// TIA Portal project "MP2019" (V17)

(* hardware
DEVICE "S7-1200 station_1"  S7-1200 Station
   slot 0: "Rack_0"  S7-1200 Rack  Rack  V1.0
   slot 1: "PLC_1"  CPU 1214C DC/DC/DC  6ES7 214-1AG40-0XB0  V4.5
*)

// ===== PLC "PLC_1"  CPU 1214C DC/DC/DC =====

VAR_GLOBAL   // PLC tag table "Default tag table"
   "wysoki_poziom" AT %I0.1 : Bool;
   "Tag_2" AT %I0.2 : Bool;
   "pompa_1" AT %Q0.0 : Bool;
   "pompa_2" AT %Q0.1 : Bool;
   "Tag_5" AT %M50.0 : Bool;
   "Tag_6" AT %M50.1 : Bool;
   "Tag_7" AT %M50.2 : Bool;
   "Tag_8" AT %M50.3 : Bool;
   "niski_poziom" AT %I0.0 : Bool;
   "Tag_10" AT %Q0.3 : Bool;
   "Tag_11" AT %I0.3 : Bool;
   "Tag_12" AT %Q0.4 : Bool;
   "Tag_13" AT %Q0.5 : Bool;
   "Tag_14" AT %Q0.6 : Bool;
   "Tag_15" AT %IW64 : Int;
   "Clock_Byte" AT %MB0 : Byte;
   "Clock_10Hz" AT %M0.0 : Bool;
   "Clock_5Hz" AT %M0.1 : Bool;
   "Clock_2.5Hz" AT %M0.2 : Bool;
   "Clock_2Hz" AT %M0.3 : Bool;
   "Clock_1.25Hz" AT %M0.4 : Bool;
   "Clock_1Hz" AT %M0.5 : Bool;
   "Clock_0.625Hz" AT %M0.6 : Bool;
   "Clock_0.5Hz" AT %M0.7 : Bool;
   "alarm" AT %Q0.7 : Bool;
   "Tag_1" AT %I0.7 : Bool;
END_VAR

DATA_BLOCK "grupowe1_DB"   // DB1
{ S7_Optimized_Access := 'TRUE' }
VERSION : 0.1
// stored: InstanceOfName grupowe1
"grupowe1"
BEGIN
END_DATA_BLOCK

DATA_BLOCK "grupowe2_DB"   // DB2
{ S7_Optimized_Access := 'TRUE' }
VERSION : 0.1
// stored: InstanceOfName grupowe2
"grupowe2"
BEGIN
END_DATA_BLOCK

DATA_BLOCK "grupowe4_DB"   // DB8
{ S7_Optimized_Access := 'TRUE' }
VERSION : 0.1
// stored: InstanceOfName grupowe4
"grupowe4"
BEGIN
END_DATA_BLOCK

DATA_BLOCK "grupowe6_DB"   // DB9
{ S7_Optimized_Access := 'TRUE' }
VERSION : 0.1
// stored: InstanceOfName grupowe6
"grupowe6"
BEGIN
END_DATA_BLOCK

DATA_BLOCK "grupowe7_DB"   // DB13
{ S7_Optimized_Access := 'TRUE' }
VERSION : 0.1
// stored: InstanceOfName grupowe7
"grupowe7"
BEGIN
END_DATA_BLOCK

DATA_BLOCK "final_Master_DB"   // DB14
{ S7_Optimized_Access := 'TRUE' }
VERSION : 0.1
// stored: InstanceOfName final_Master
"final_Master"
BEGIN
END_DATA_BLOCK

DATA_BLOCK "final_Ekspert_DB"   // DB15
{ S7_Optimized_Access := 'TRUE' }
VERSION : 0.1
// stored: InstanceOfName final_Ekspert
"final_Ekspert"
BEGIN
END_DATA_BLOCK

// folder: System blocks/Program resources

DATA_BLOCK "IEC_Timer_0_DB"   // DB3
{ S7_Optimized_Access := 'TRUE' }
AUTHOR : Simatic
FAMILY : IEC
NAME : IEC_TMR
VERSION : 1.0
// stored: InstanceOfName IEC_TIMER
"IEC_TIMER"
BEGIN
END_DATA_BLOCK

DATA_BLOCK "IEC_Timer_0_DB_1"   // DB4
{ S7_Optimized_Access := 'TRUE' }
AUTHOR : Simatic
FAMILY : IEC
NAME : IEC_TMR
VERSION : 1.0
// stored: InstanceOfName IEC_TIMER
"IEC_TIMER"
BEGIN
END_DATA_BLOCK

DATA_BLOCK "Counter0"   // DB5
{ S7_Optimized_Access := 'TRUE' }
AUTHOR : Simatic
FAMILY : IEC
NAME : CNTR
VERSION : 1.0
// stored: InstanceOfName IEC_COUNTER
"IEC_COUNTER"
BEGIN
END_DATA_BLOCK

DATA_BLOCK "IEC_Timer_0_DB_3"   // DB6
{ S7_Optimized_Access := 'TRUE' }
AUTHOR : Simatic
FAMILY : IEC
NAME : IEC_TMR
VERSION : 1.0
// stored: InstanceOfName IEC_TIMER
"IEC_TIMER"
BEGIN
END_DATA_BLOCK

DATA_BLOCK "IEC_Timer_0_DB_4"   // DB7
{ S7_Optimized_Access := 'TRUE' }
AUTHOR : Simatic
FAMILY : IEC
NAME : IEC_TMR
VERSION : 1.0
// stored: InstanceOfName IEC_TIMER
"IEC_TIMER"
BEGIN
END_DATA_BLOCK

DATA_BLOCK "TON0"   // DB10
{ S7_Optimized_Access := 'TRUE' }
AUTHOR : Simatic
FAMILY : IEC
NAME : IEC_TMR
VERSION : 1.0
// stored: InstanceOfName IEC_TIMER
"IEC_TIMER"
BEGIN
END_DATA_BLOCK

DATA_BLOCK "TON1"   // DB11
{ S7_Optimized_Access := 'TRUE' }
AUTHOR : Simatic
FAMILY : IEC
NAME : IEC_TMR
VERSION : 1.0
// stored: InstanceOfName IEC_TIMER
"IEC_TIMER"
BEGIN
END_DATA_BLOCK

DATA_BLOCK "TON2"   // DB12
{ S7_Optimized_Access := 'TRUE' }
AUTHOR : Simatic
FAMILY : IEC
NAME : IEC_TMR
VERSION : 1.0
// stored: InstanceOfName IEC_TIMER
"IEC_TIMER"
BEGIN
END_DATA_BLOCK

// folder: (top level)

FUNCTION_BLOCK "grupowe1"   // FB1, LAD
{ S7_Optimized_Access := 'TRUE' }
VERSION : 0.1
   VAR_INPUT
      IN1 : Bool;
      IN2 : Bool;
   END_VAR
   VAR_IN_OUT
      OUT0 : Bool;
      OUT1 : Bool;
   END_VAR
   VAR
      IN1_edge : Bool;
      IN2_edge : Bool;
   END_VAR
   VAR_TEMP
      prev_OUT0 : Bool;
      prev_OUT1 : Bool;
   END_VAR
   VAR_TEMP   // added for the SCL form of the ladder/FBD networks
      _w1 : Bool;
   END_VAR
BEGIN

REGION Network 1
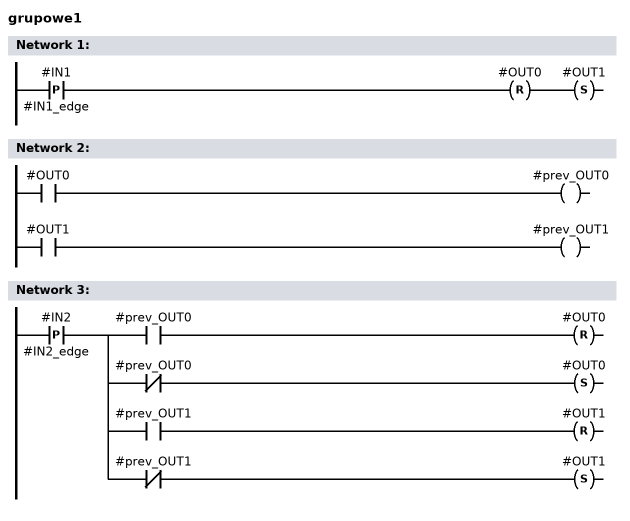
   RUNG wire#powerrail
      P_Contact(operand := #IN1, bit := #IN1_edge)
      R_Coil( #OUT0 )
      S_Coil( #OUT1 )
   END_RUNG
   // the same network as SCL:
   #_w1 := #IN1 AND NOT #IN1_edge;   // rising edge of #IN1
   #IN1_edge := #IN1;
   IF #_w1 THEN
       #OUT0 := FALSE;
       #OUT1 := TRUE;
   END_IF;
END_REGION

REGION Network 2
   RUNG wire#powerrail
      Contact( #OUT0 )
      Coil( #prev_OUT0 )
   END_RUNG
   RUNG wire#powerrail
      Contact( #OUT1 )
      Coil( #prev_OUT1 )
   END_RUNG
   // the same network as SCL:
   #prev_OUT0 := #OUT0;
   #prev_OUT1 := #OUT1;
END_REGION

REGION Network 3
   RUNG wire#powerrail
      P_Contact(operand := #IN2, bit := #IN2_edge)
      wire#w1
      Contact( #prev_OUT0 )
      R_Coil( #OUT0 )
   END_RUNG
   RUNG wire#w1
      I_Contact( #prev_OUT0 )
      S_Coil( #OUT0 )
   END_RUNG
   RUNG wire#w1
      Contact( #prev_OUT1 )
      R_Coil( #OUT1 )
   END_RUNG
   RUNG wire#w1
      I_Contact( #prev_OUT1 )
      S_Coil( #OUT1 )
   END_RUNG
   // the same network as SCL:
   #_w1 := #IN2 AND NOT #IN2_edge;   // rising edge of #IN2
   #IN2_edge := #IN2;
   IF #_w1 AND #prev_OUT0 THEN #OUT0 := FALSE; END_IF;
   IF #_w1 AND NOT #prev_OUT0 THEN #OUT0 := TRUE; END_IF;
   IF #_w1 AND #prev_OUT1 THEN #OUT1 := FALSE; END_IF;
   IF #_w1 AND NOT #prev_OUT1 THEN #OUT1 := TRUE; END_IF;
END_REGION
END_FUNCTION_BLOCK

FUNCTION_BLOCK "grupowe2"   // FB2, LAD
{ S7_Optimized_Access := 'TRUE' }
VERSION : 0.1
   VAR_INPUT
      IN2 : Bool;
      IN3 : Bool;
   END_VAR
   VAR_IN_OUT
      OUT3 : Bool;
   END_VAR
   VAR
      IN2_edge : Bool;
      IN3_edge : Bool;
      step1 : Bool;
   END_VAR
   VAR_TEMP
      prev_OUT3 : Bool;
   END_VAR
   VAR_TEMP   // added for the SCL form of the ladder/FBD networks
      _w1 : Bool;
      _w2 : Bool;
   END_VAR
BEGIN

REGION Network 1
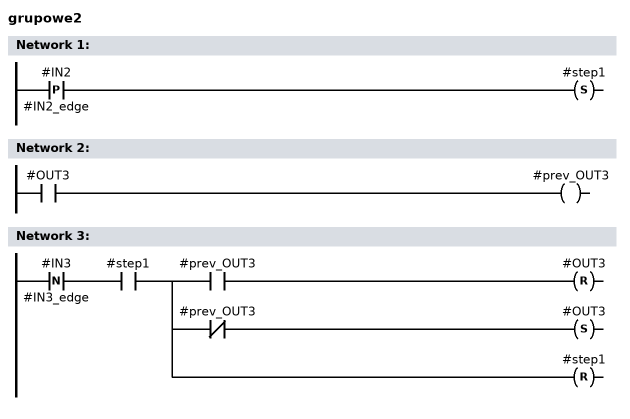
   RUNG wire#powerrail
      P_Contact(operand := #IN2, bit := #IN2_edge)
      S_Coil( #step1 )
   END_RUNG
   // the same network as SCL:
   #_w1 := #IN2 AND NOT #IN2_edge;   // rising edge of #IN2
   #IN2_edge := #IN2;
   IF #_w1 THEN #step1 := TRUE; END_IF;
END_REGION

REGION Network 2
   RUNG wire#powerrail
      Contact( #OUT3 )
      Coil( #prev_OUT3 )
   END_RUNG
   // the same network as SCL:
   #prev_OUT3 := #OUT3;
END_REGION

REGION Network 3
   RUNG wire#powerrail
      N_Contact(operand := #IN3, bit := #IN3_edge)
      Contact( #step1 )
      wire#w1
      Contact( #prev_OUT3 )
      R_Coil( #OUT3 )
   END_RUNG
   RUNG wire#w1
      I_Contact( #prev_OUT3 )
      S_Coil( #OUT3 )
   END_RUNG
   RUNG wire#w1
      R_Coil( #step1 )
   END_RUNG
   // the same network as SCL:
   #_w1 := NOT #IN3 AND #IN3_edge;   // falling edge of #IN3
   #IN3_edge := #IN3;
   #_w2 := #_w1 AND #step1;
   IF #_w2 AND #prev_OUT3 THEN #OUT3 := FALSE; END_IF;
   IF #_w2 AND NOT #prev_OUT3 THEN #OUT3 := TRUE; END_IF;
   IF #_w2 THEN #step1 := FALSE; END_IF;
END_REGION
END_FUNCTION_BLOCK

FUNCTION_BLOCK "grupowe4"   // FB3, LAD
{ S7_Optimized_Access := 'TRUE' }
VERSION : 0.1
   VAR_INPUT
      IN2 : Bool;
   END_VAR
   VAR_OUTPUT
      OUT : Bool;
   END_VAR
BEGIN

REGION Network 1
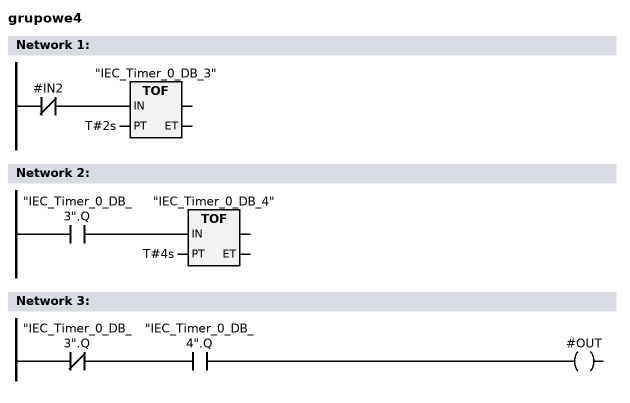
   "IEC_Timer_0_DB_3".TOF(IN := NOT #IN2, PT := T#2s);
END_REGION

REGION Network 2
   "IEC_Timer_0_DB_4".TOF(IN := "IEC_Timer_0_DB_3".Q, PT := T#4s);
END_REGION

REGION Network 3
   RUNG wire#powerrail
      I_Contact( "IEC_Timer_0_DB_3".Q )
      Contact( "IEC_Timer_0_DB_4".Q )
      Coil( #OUT )
   END_RUNG
   // the same network as SCL:
   #OUT := NOT "IEC_Timer_0_DB_3".Q AND "IEC_Timer_0_DB_4".Q;
END_REGION
END_FUNCTION_BLOCK

FUNCTION_BLOCK "grupowe6"   // FB4, LAD
{ S7_Optimized_Access := 'TRUE' }
VERSION : 0.1
   VAR_INPUT
      IN2 : Bool;
      IN3 : Bool;
   END_VAR
   VAR_OUTPUT
      OUT0 : Bool;
   END_VAR
   VAR_IN_OUT
      Value : Int;
   END_VAR
   VAR
      IN2_edge : Bool;
      IN3_edge : Bool;
   END_VAR
   VAR_TEMP
      Modulo : USInt;
   END_VAR
   VAR_TEMP   // added for the SCL form of the ladder/FBD networks
      _w1 : Bool;
      _w2 : Bool;
   END_VAR
BEGIN

REGION Network 1
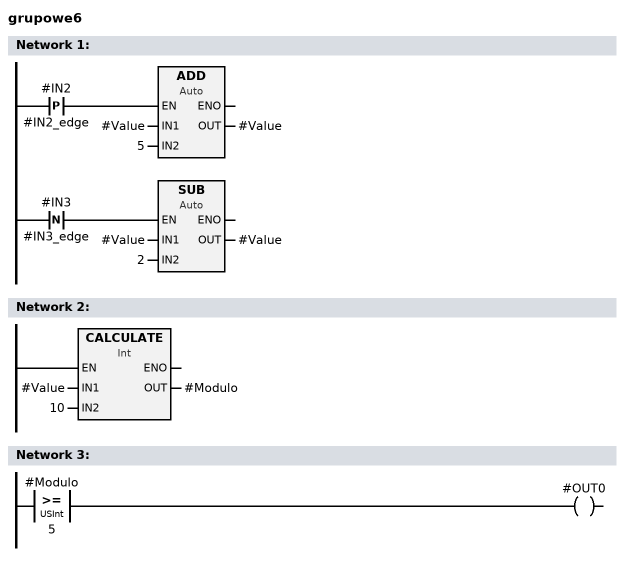
   RUNG wire#powerrail
      P_Contact(operand := #IN2, bit := #IN2_edge)
      Add(in1 := #Value, in2 := 5, out => #Value)
   END_RUNG
   RUNG wire#powerrail
      N_Contact(operand := #IN3, bit := #IN3_edge)
      Sub(in1 := #Value, in2 := 2, out => #Value)
   END_RUNG
   // the same network as SCL:
   #_w1 := #IN2 AND NOT #IN2_edge;   // rising edge of #IN2
   #IN2_edge := #IN2;
   IF #_w1 THEN #Value := #Value + 5; END_IF;
   #_w2 := NOT #IN3 AND #IN3_edge;   // falling edge of #IN3
   #IN3_edge := #IN3;
   IF #_w2 THEN #Value := #Value - 2; END_IF;
END_REGION

REGION Network 2
   RUNG wire#powerrail
      { S7_Templates := "SrcType := Int"; S7_Expression := "IN1 MOD IN2" } Calculate(in1 := #Value, in2 := 10, out => #Modulo)
   END_RUNG
   // the same network as SCL:
   #Modulo := #Value MOD 10;
END_REGION

REGION Network 3
   RUNG wire#powerrail
      { S7_Templates := "SrcType := USInt" } GE_Contact(in1 := #Modulo, in2 := 5)
      Coil( #OUT0 )
   END_RUNG
   // the same network as SCL:
   #OUT0 := #Modulo >= 5;
END_REGION
END_FUNCTION_BLOCK

FUNCTION_BLOCK "grupowe7"   // FB5, LAD
{ S7_Optimized_Access := 'TRUE' }
VERSION : 0.1
   VAR_INPUT
      Analog_signal : Int;
   END_VAR
   VAR_OUTPUT
      OUT0 : Bool;
      OUT4 : Bool;
      OUT5 : Bool;
      OUT6 : Bool;
   END_VAR
   VAR
      TON0_Q : Bool;
   END_VAR
   VAR_TEMP
      duty : Int;
      Analog_norm : Real;
      T_high : DInt;
      Hz : Bool;
   END_VAR
BEGIN

REGION Network 1
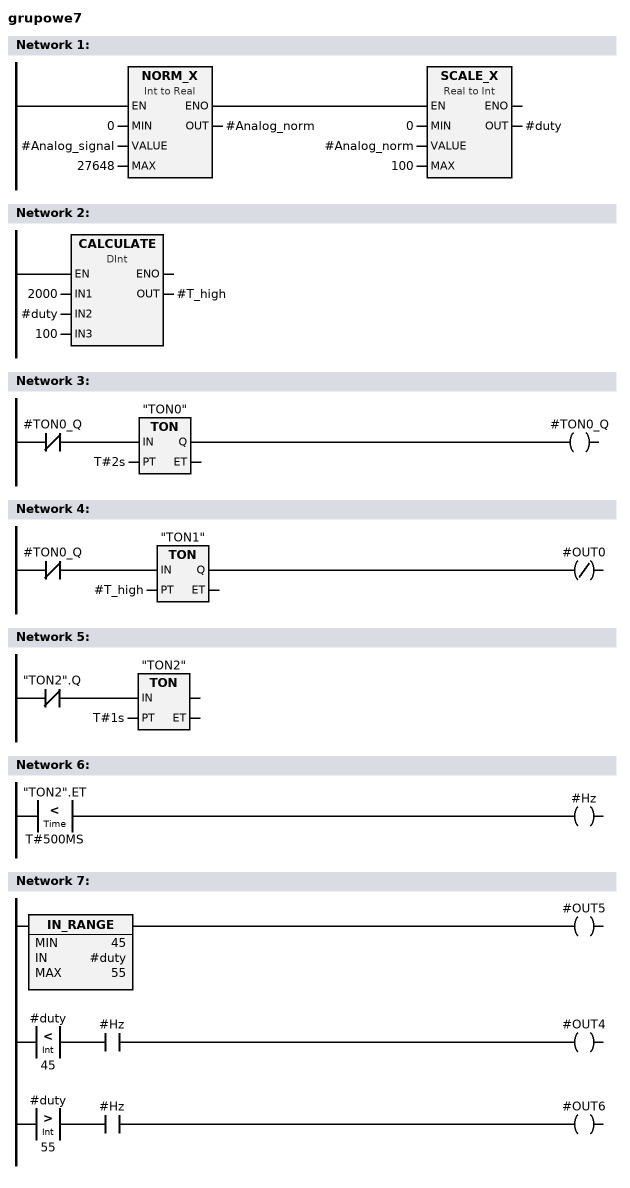
   RUNG wire#powerrail
      { S7_Templates := "[SrcType := Int, DestType := Real]" } Normalize(min := 0, value := #Analog_signal, max := 27648, out => #Analog_norm)
      { S7_Templates := "[SrcType := Real, DestType := Int]" } Scale(min := 0, value := #Analog_norm, max := 100, out => #duty)
   END_RUNG
   // the same network as SCL:
   #Analog_norm := NORM_X(MIN := 0, VALUE := #Analog_signal, MAX := 27648);
   #duty := SCALE_X(MIN := 0, VALUE := #Analog_norm, MAX := 100);
END_REGION

REGION Network 2
   RUNG wire#powerrail
      { S7_Templates := "SrcType := DInt"; S7_Expression := "IN1 * IN2 / IN3" } Calculate(in1 := 2000, in2 := #duty, in3 := 100, out => #T_high)
   END_RUNG
   // the same network as SCL:
   #T_high := 2000 * #duty / 100;
END_REGION

REGION Network 3
   "TON0".TON(IN := NOT #TON0_Q, PT := T#2s);
   #TON0_Q := "TON0".Q;
END_REGION

REGION Network 4
   "TON1".TON(IN := NOT #TON0_Q, PT := #T_high);
   #OUT0 := NOT "TON1".Q;
END_REGION

REGION Network 5
   "TON2".TON(IN := NOT "TON2".Q, PT := T#1s);
END_REGION

REGION Network 6
   RUNG wire#powerrail
      { S7_Templates := "SrcType := Time" } LT_Contact(in1 := "TON2".ET, in2 := T#500MS)
      Coil( #Hz )
   END_RUNG
   // the same network as SCL:
   #Hz := "TON2".ET < T#500MS;
END_REGION

REGION Network 7
   RUNG wire#powerrail
      { S7_Templates := "SrcType := Int" } InRange(min := 45, in := #duty, max := 55)
      Coil( #OUT5 )
   END_RUNG
   RUNG wire#powerrail
      { S7_Templates := "SrcType := Int" } LT_Contact(in1 := #duty, in2 := 45)
      Contact( #Hz )
      Coil( #OUT4 )
   END_RUNG
   RUNG wire#powerrail
      { S7_Templates := "SrcType := Int" } GT_Contact(in1 := #duty, in2 := 55)
      Contact( #Hz )
      Coil( #OUT6 )
   END_RUNG
   // the same network as SCL:
   #OUT5 := (45 <= #duty) AND (#duty <= 55);
   #OUT4 := (#duty < 45) AND #Hz;
   #OUT6 := (#duty > 55) AND #Hz;
END_REGION
END_FUNCTION_BLOCK

FUNCTION_BLOCK "final_Master"   // FB6, LAD
{ S7_Optimized_Access := 'TRUE' }
VERSION : 0.1
   VAR_INPUT
      niski_poziom : Bool;
      wysoki_poziom : Bool;
   END_VAR
   VAR_OUTPUT
      alarm : Bool;
      segment1 : Bool;
      segment2 : Bool;
      segment4 : Bool;
   END_VAR
   VAR_IN_OUT
      pompa_1 : Bool;
      pompa_2 : Bool;
   END_VAR
   VAR
      niski_zbocze : Bool;
      wysoki_zbocze : Bool;
      pompa_ostatnio : Bool;
      niski_zbocze2 : Bool;
      wysoki_zbocze2 : Bool;
      prev_pompa : Bool;
   END_VAR
   VAR_TEMP   // added for the SCL form of the ladder/FBD networks
      _w1 : Bool;
      _w2 : Bool;
      _w3 : Bool;
   END_VAR
BEGIN

REGION Network 1
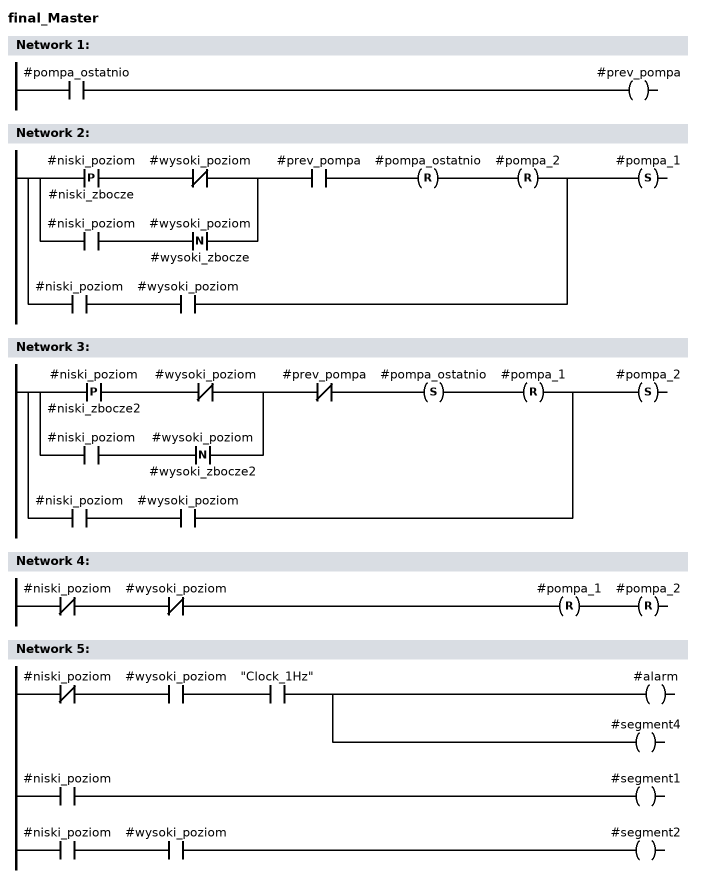
   RUNG wire#powerrail
      Contact( #pompa_ostatnio )
      Coil( #prev_pompa )
   END_RUNG
   // the same network as SCL:
   #prev_pompa := #pompa_ostatnio;
END_REGION

REGION Network 2
   RUNG wire#powerrail
      P_Contact(operand := #niski_poziom, bit := #niski_zbocze)
      I_Contact( #wysoki_poziom )
      wire#w1
      Contact( #prev_pompa )
      R_Coil( #pompa_ostatnio )
      R_Coil( #pompa_2 )
      wire#w2
      S_Coil( #pompa_1 )
   END_RUNG
   RUNG wire#powerrail
      Contact( #niski_poziom )
      N_Contact(operand := #wysoki_poziom, bit := #wysoki_zbocze)
   END_RUNG wire#w1
   RUNG wire#powerrail
      Contact( #niski_poziom )
      Contact( #wysoki_poziom )
   END_RUNG wire#w2
   // the same network as SCL:
   #_w1 := #niski_poziom AND NOT #niski_zbocze;   // rising edge of #niski_poziom
   #niski_zbocze := #niski_poziom;
   #_w2 := #niski_poziom AND NOT #wysoki_poziom AND #wysoki_zbocze;   // falling edge of #wysoki_poziom
   #wysoki_zbocze := #wysoki_poziom;
   #_w3 := ((#_w1 AND NOT #wysoki_poziom) OR #_w2) AND #prev_pompa;
   IF #_w3 THEN
       #pompa_ostatnio := FALSE;
       #pompa_2 := FALSE;
   END_IF;
   IF #_w3 OR (#niski_poziom AND #wysoki_poziom) THEN #pompa_1 := TRUE; END_IF;
END_REGION

REGION Network 3
   RUNG wire#powerrail
      P_Contact(operand := #niski_poziom, bit := #niski_zbocze2)
      I_Contact( #wysoki_poziom )
      wire#w1
      I_Contact( #prev_pompa )
      S_Coil( #pompa_ostatnio )
      R_Coil( #pompa_1 )
      wire#w2
      S_Coil( #pompa_2 )
   END_RUNG
   RUNG wire#powerrail
      Contact( #niski_poziom )
      N_Contact(operand := #wysoki_poziom, bit := #wysoki_zbocze2)
   END_RUNG wire#w1
   RUNG wire#powerrail
      Contact( #niski_poziom )
      Contact( #wysoki_poziom )
   END_RUNG wire#w2
   // the same network as SCL:
   #_w1 := #niski_poziom AND NOT #niski_zbocze2;   // rising edge of #niski_poziom
   #niski_zbocze2 := #niski_poziom;
   #_w2 := #niski_poziom AND NOT #wysoki_poziom AND #wysoki_zbocze2;   // falling edge of #wysoki_poziom
   #wysoki_zbocze2 := #wysoki_poziom;
   #_w3 := ((#_w1 AND NOT #wysoki_poziom) OR #_w2) AND NOT #prev_pompa;
   IF #_w3 THEN
       #pompa_ostatnio := TRUE;
       #pompa_1 := FALSE;
   END_IF;
   IF #_w3 OR (#niski_poziom AND #wysoki_poziom) THEN #pompa_2 := TRUE; END_IF;
END_REGION

REGION Network 4
   RUNG wire#powerrail
      I_Contact( #niski_poziom )
      I_Contact( #wysoki_poziom )
      R_Coil( #pompa_1 )
      R_Coil( #pompa_2 )
   END_RUNG
   // the same network as SCL:
   IF NOT #niski_poziom AND NOT #wysoki_poziom THEN
       #pompa_1 := FALSE;
       #pompa_2 := FALSE;
   END_IF;
END_REGION

REGION Network 5
   RUNG wire#powerrail
      I_Contact( #niski_poziom )
      Contact( #wysoki_poziom )
      Contact( "Clock_1Hz" )
      wire#w1
      Coil( #alarm )
   END_RUNG
   RUNG wire#w1
      Coil( #segment4 )
   END_RUNG
   RUNG wire#powerrail
      Contact( #niski_poziom )
      Coil( #segment1 )
   END_RUNG
   RUNG wire#powerrail
      Contact( #niski_poziom )
      Contact( #wysoki_poziom )
      Coil( #segment2 )
   END_RUNG
   // the same network as SCL:
   #alarm := NOT #niski_poziom AND #wysoki_poziom AND "Clock_1Hz";
   #segment4 := #alarm;
   #segment1 := #niski_poziom;
   #segment2 := #niski_poziom AND #wysoki_poziom;
END_REGION
END_FUNCTION_BLOCK

FUNCTION_BLOCK "final_Ekspert"   // FB7, LAD
{ S7_Optimized_Access := 'TRUE' }
VERSION : 0.1
   VAR_INPUT
      niski_poziom : Bool;
      wysoki_poziom : Bool;
      tryb_pracy_zmiana : Bool;
   END_VAR
   VAR_OUTPUT
      alarm : Bool;
      segment1 : Bool;
      segment2 : Bool;
      segment4 : Bool;
   END_VAR
   VAR_IN_OUT
      pompa_1 : Bool;
      tryb_pracy : Int;
      pompa_2 : Bool;
   END_VAR
   VAR
      niski_zbocze : Bool;
      wysoki_zbocze : Bool;
      pompa_ostatnio : Bool;
      niski_zbocze2 : Bool;
      wysoki_zbocze2 : Bool;
      prev_pompa : Bool;
      tryb_pracy_zboczeP : Bool;
      tryb_pracy_zboczeN : Bool;
   END_VAR
   VAR_TEMP   // added for the SCL form of the ladder/FBD networks
      _w1 : Bool;
      _w2 : Bool;
      _w3 : Bool;
      _w4 : Bool;
   END_VAR
BEGIN

REGION Network 1
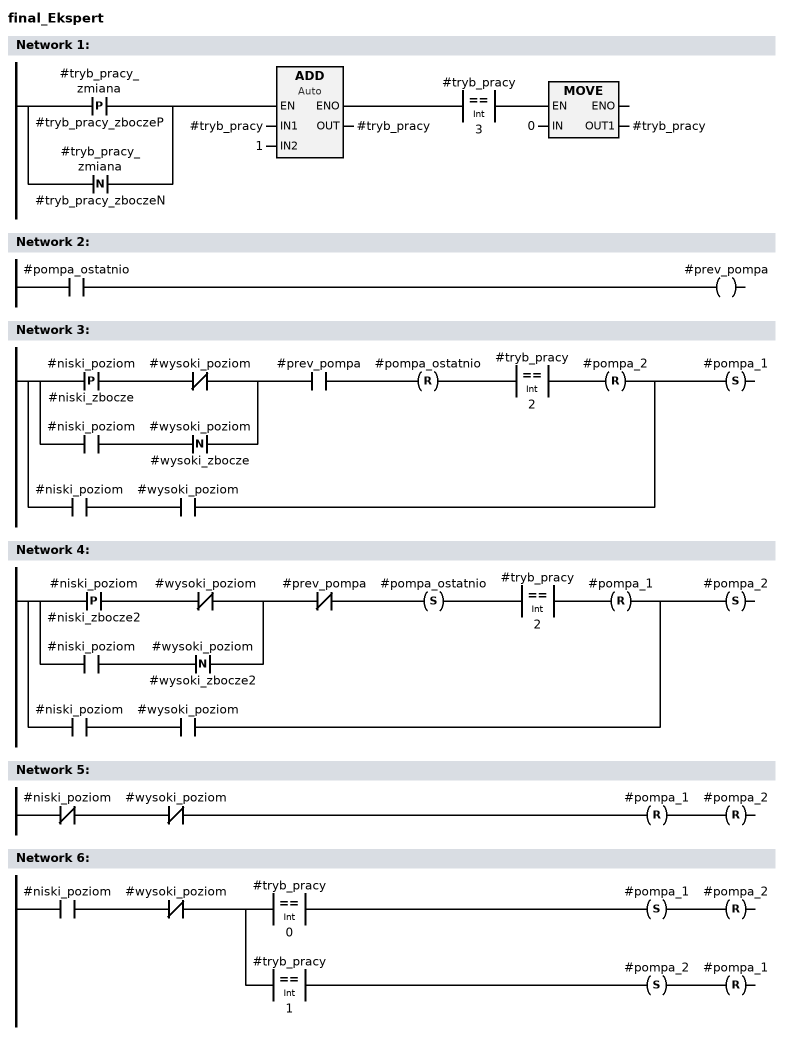
   RUNG wire#powerrail
      P_Contact(operand := #tryb_pracy_zmiana, bit := #tryb_pracy_zboczeP)
      wire#w1
      Add(in1 := #tryb_pracy, in2 := 1, out => #tryb_pracy)
      { S7_Templates := "SrcType := Int" } EQ_Contact(in1 := #tryb_pracy, in2 := 3)
      Move(in := 0, out1 => #tryb_pracy)
   END_RUNG
   RUNG wire#powerrail
      N_Contact(operand := #tryb_pracy_zmiana, bit := #tryb_pracy_zboczeN)
   END_RUNG wire#w1
   // the same network as SCL:
   #_w1 := #tryb_pracy_zmiana AND NOT #tryb_pracy_zboczeP;   // rising edge of #tryb_pracy_zmiana
   #tryb_pracy_zboczeP := #tryb_pracy_zmiana;
   #_w2 := NOT #tryb_pracy_zmiana AND #tryb_pracy_zboczeN;   // falling edge of #tryb_pracy_zmiana
   #tryb_pracy_zboczeN := #tryb_pracy_zmiana;
   #_w3 := #_w1 OR #_w2;
   IF #_w3 THEN #tryb_pracy := #tryb_pracy + 1; END_IF;
   IF #_w3 AND (#tryb_pracy = 3) THEN #tryb_pracy := 0; END_IF;
END_REGION

REGION Network 2
   RUNG wire#powerrail
      Contact( #pompa_ostatnio )
      Coil( #prev_pompa )
   END_RUNG
   // the same network as SCL:
   #prev_pompa := #pompa_ostatnio;
END_REGION

REGION Network 3
   RUNG wire#powerrail
      P_Contact(operand := #niski_poziom, bit := #niski_zbocze)
      I_Contact( #wysoki_poziom )
      wire#w1
      Contact( #prev_pompa )
      R_Coil( #pompa_ostatnio )
      { S7_Templates := "SrcType := Int" } EQ_Contact(in1 := #tryb_pracy, in2 := 2)
      R_Coil( #pompa_2 )
      wire#w2
      S_Coil( #pompa_1 )
   END_RUNG
   RUNG wire#powerrail
      Contact( #niski_poziom )
      N_Contact(operand := #wysoki_poziom, bit := #wysoki_zbocze)
   END_RUNG wire#w1
   RUNG wire#powerrail
      Contact( #niski_poziom )
      Contact( #wysoki_poziom )
   END_RUNG wire#w2
   // the same network as SCL:
   #_w1 := #niski_poziom AND NOT #niski_zbocze;   // rising edge of #niski_poziom
   #niski_zbocze := #niski_poziom;
   #_w2 := #niski_poziom AND NOT #wysoki_poziom AND #wysoki_zbocze;   // falling edge of #wysoki_poziom
   #wysoki_zbocze := #wysoki_poziom;
   #_w3 := ((#_w1 AND NOT #wysoki_poziom) OR #_w2) AND #prev_pompa;
   IF #_w3 THEN #pompa_ostatnio := FALSE; END_IF;
   #_w4 := #_w3 AND (#tryb_pracy = 2);
   IF #_w4 THEN #pompa_2 := FALSE; END_IF;
   IF #_w4 OR (#niski_poziom AND #wysoki_poziom) THEN #pompa_1 := TRUE; END_IF;
END_REGION

REGION Network 4
   RUNG wire#powerrail
      P_Contact(operand := #niski_poziom, bit := #niski_zbocze2)
      I_Contact( #wysoki_poziom )
      wire#w1
      I_Contact( #prev_pompa )
      S_Coil( #pompa_ostatnio )
      { S7_Templates := "SrcType := Int" } EQ_Contact(in1 := #tryb_pracy, in2 := 2)
      R_Coil( #pompa_1 )
      wire#w2
      S_Coil( #pompa_2 )
   END_RUNG
   RUNG wire#powerrail
      Contact( #niski_poziom )
      N_Contact(operand := #wysoki_poziom, bit := #wysoki_zbocze2)
   END_RUNG wire#w1
   RUNG wire#powerrail
      Contact( #niski_poziom )
      Contact( #wysoki_poziom )
   END_RUNG wire#w2
   // the same network as SCL:
   #_w1 := #niski_poziom AND NOT #niski_zbocze2;   // rising edge of #niski_poziom
   #niski_zbocze2 := #niski_poziom;
   #_w2 := #niski_poziom AND NOT #wysoki_poziom AND #wysoki_zbocze2;   // falling edge of #wysoki_poziom
   #wysoki_zbocze2 := #wysoki_poziom;
   #_w3 := ((#_w1 AND NOT #wysoki_poziom) OR #_w2) AND NOT #prev_pompa;
   IF #_w3 THEN #pompa_ostatnio := TRUE; END_IF;
   #_w4 := #_w3 AND (#tryb_pracy = 2);
   IF #_w4 THEN #pompa_1 := FALSE; END_IF;
   IF #_w4 OR (#niski_poziom AND #wysoki_poziom) THEN #pompa_2 := TRUE; END_IF;
END_REGION

REGION Network 5
   RUNG wire#powerrail
      I_Contact( #niski_poziom )
      I_Contact( #wysoki_poziom )
      R_Coil( #pompa_1 )
      R_Coil( #pompa_2 )
   END_RUNG
   // the same network as SCL:
   IF NOT #niski_poziom AND NOT #wysoki_poziom THEN
       #pompa_1 := FALSE;
       #pompa_2 := FALSE;
   END_IF;
END_REGION

REGION Network 6
   RUNG wire#powerrail
      Contact( #niski_poziom )
      I_Contact( #wysoki_poziom )
      wire#w1
      { S7_Templates := "SrcType := Int" } EQ_Contact(in1 := #tryb_pracy, in2 := 0)
      S_Coil( #pompa_1 )
      R_Coil( #pompa_2 )
   END_RUNG
   RUNG wire#w1
      { S7_Templates := "SrcType := Int" } EQ_Contact(in1 := #tryb_pracy, in2 := 1)
      S_Coil( #pompa_2 )
      R_Coil( #pompa_1 )
   END_RUNG
   // the same network as SCL:
   #_w1 := #niski_poziom AND NOT #wysoki_poziom;
   IF #_w1 AND (#tryb_pracy = 0) THEN
       #pompa_1 := TRUE;
       #pompa_2 := FALSE;
   END_IF;
   IF #_w1 AND (#tryb_pracy = 1) THEN
       #pompa_2 := TRUE;
       #pompa_1 := FALSE;
   END_IF;
END_REGION
END_FUNCTION_BLOCK

FUNCTION "grupowe3" : Void   // FC1, LAD
{ S7_Optimized_Access := 'TRUE' }
VERSION : 0.1
   VAR_INPUT
      f : Real;
      duty : Int;
   END_VAR
   VAR_OUTPUT
      OUT : Bool;
   END_VAR
   VAR_TEMP
      T : DInt;
      T_Real : Real;
      T_high : DInt;
   END_VAR
BEGIN

REGION Network 1
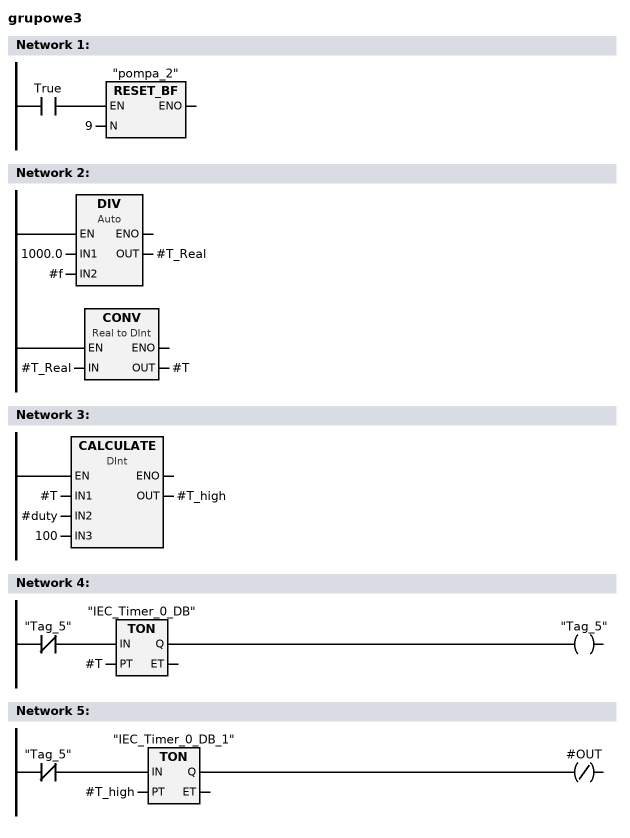
   // no SCL statement known for RBitfield: written as a call
   IF True THEN RESET_BF(operand := "pompa_2", n := 9); END_IF;
END_REGION

REGION Network 2
   RUNG wire#powerrail
      Div(in1 := 1000.0, in2 := #f, out => #T_Real)
   END_RUNG
   RUNG wire#powerrail
      { S7_Templates := "[SrcType := Real, DestType := DInt]" } Convert(in := #T_Real, out => #T)
   END_RUNG
   // the same network as SCL:
   #T_Real := 1000.0 / #f;
   #T := REAL_TO_DINT(#T_Real);
END_REGION

REGION Network 3
   RUNG wire#powerrail
      { S7_Templates := "SrcType := DInt"; S7_Expression := "IN1*IN2/IN3" } Calculate(in1 := #T, in2 := #duty, in3 := 100, out => #T_high)
   END_RUNG
   // the same network as SCL:
   #T_high := #T*#duty/100;
END_REGION

REGION Network 4
   "IEC_Timer_0_DB".TON(IN := NOT "Tag_5", PT := #T);
   "Tag_5" := "IEC_Timer_0_DB".Q;
END_REGION

REGION Network 5
   "IEC_Timer_0_DB_1".TON(IN := NOT "Tag_5", PT := #T_high);
   #OUT := NOT "IEC_Timer_0_DB_1".Q;
END_REGION
END_FUNCTION

FUNCTION "grupowe5" : Void   // FC2, LAD
{ S7_Optimized_Access := 'TRUE' }
VERSION : 0.1
   VAR_INPUT
      IN : Bool;
   END_VAR
   VAR_OUTPUT
      OUT : Bool;
   END_VAR
   VAR_TEMP
      Mod_result : Int;
   END_VAR
BEGIN

REGION Network 1
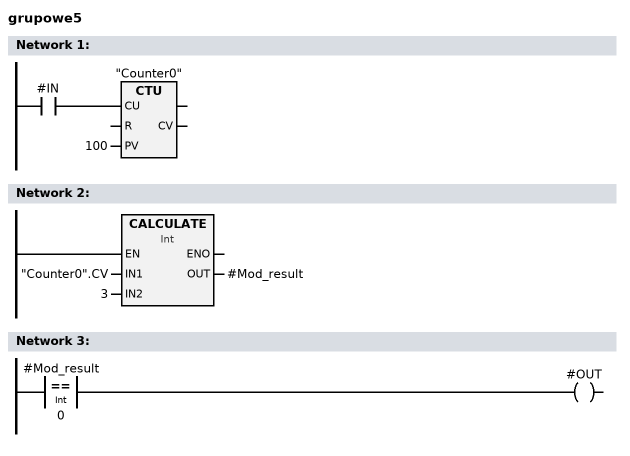
   "Counter0".CTU(CU := #IN, PV := 100);
END_REGION

REGION Network 2
   RUNG wire#powerrail
      { S7_Templates := "SrcType := Int"; S7_Expression := "IN1 MOD IN2" } Calculate(in1 := "Counter0".CV, in2 := 3, out => #Mod_result)
   END_RUNG
   // the same network as SCL:
   #Mod_result := "Counter0".CV MOD 3;
END_REGION

REGION Network 3
   RUNG wire#powerrail
      { S7_Templates := "SrcType := Int" } EQ_Contact(in1 := #Mod_result, in2 := 0)
      Coil( #OUT )
   END_RUNG
   // the same network as SCL:
   #OUT := #Mod_result = 0;
END_REGION
END_FUNCTION

ORGANIZATION_BLOCK "Main"   // OB1, LAD, ProgramCycle
TITLE = "Main Program Sweep (Cycle)"
{ S7_Optimized_Access := 'TRUE' }
VERSION : 0.1
   VAR_INPUT
      Initial_Call : Bool;   // Initial call of this OB
      Remanence : Bool;   // =True, if remanent data are available
   END_VAR
BEGIN

REGION Network 1
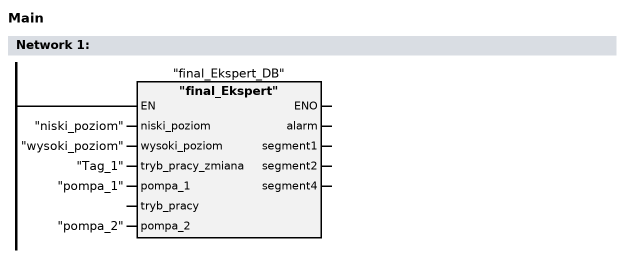
   RUNG wire#powerrail
      "final_Ekspert_DB"(niski_poziom := "niski_poziom", wysoki_poziom := "wysoki_poziom", tryb_pracy_zmiana := "Tag_1", pompa_1 := "pompa_1", tryb_pracy :=, pompa_2 := "pompa_2", alarm =>, segment1 =>, segment2 =>, segment4 =>)
   END_RUNG
   // the same network as SCL:
   "final_Ekspert_DB"(niski_poziom := "niski_poziom",   // "final_Ekspert"
                      wysoki_poziom := "wysoki_poziom",
                      tryb_pracy_zmiana := "Tag_1",
                      pompa_1 := "pompa_1",
                      pompa_2 := "pompa_2");
END_REGION
END_ORGANIZATION_BLOCK